PROGRAM POU
VAR
    fbDALI102Off             : FB_DALI102Off(POU_Comm.fbKL6821Communication);
    fbDALI102Off1            : FB_DALI102Off(POU_Comm.fbKL6821Communication);
    fbDALI102Off2            : FB_DALI102Off(POU_Comm.fbKL6821Communication);
    fbDALI102Off3            : FB_DALI102Off(POU_Comm.fbKL6821Communication);
    fbDALI102Dimmer1Switch   : FB_DALI102Dimmer1Switch(POU_Comm.fbKL6821Communication);
    fbDALI102Dimmer2Switch   : FB_DALI102Dimmer1Switch(POU_Comm.fbKL6821Communication);
    fbDALI102Dimmer3Switch   : FB_DALI102Dimmer1Switch(POU_Comm.fbKL6821Communication);
    fbDALI102Dimmer4Switch   : FB_DALI102Dimmer1Switch(POU_Comm.fbKL6821Communication);
    fbDALI102Dimmer5Switch   : FB_DALI102Dimmer1Switch(POU_Comm.fbKL6821Communication);
    fbDALI102Dimmer6Switch   : FB_DALI102Dimmer1Switch(POU_Comm.fbKL6821Communication);
    fbDALI102Dimmer7Switch   : FB_DALI102Dimmer1Switch(POU_Comm.fbKL6821Communication);
    fbDALI102Dimmer8Switch   : FB_DALI102Dimmer1Switch(POU_Comm.fbKL6821Communication);
    fbDALI102Dimmer9Switch   : FB_DALI102Dimmer1Switch(POU_Comm.fbKL6821Communication);
    fbDALI102Dimmer10Switch  : FB_DALI102Dimmer1Switch(POU_Comm.fbKL6821Communication);
    fbDALI102Dimmer11Switch  : FB_DALI102Dimmer1Switch(POU_Comm.fbKL6821Communication);
    fbDALI102Dimmer12Switch  : FB_DALI102Dimmer1Switch(POU_Comm.fbKL6821Communication);
    fbDALI102Dimmer13Switch  : FB_DALI102Dimmer1Switch(POU_Comm.fbKL6821Communication);
    fbDALI102Dimmer14Switch  : FB_DALI102Dimmer1Switch(POU_Comm.fbKL6821Communication);
    fbDALI102Dimmer15Switch  : FB_DALI102Dimmer1Switch(POU_Comm.fbKL6821Communication);
    fbDALI102Dimmer16Switch  : FB_DALI102Dimmer1Switch(POU_Comm.fbKL6821Communication);
    fbDALI102Dimmer17Switch  : FB_DALI102Dimmer1Switch(POU_Comm.fbKL6821Communication);
    fbDALI102Dimmer18Switch  : FB_DALI102Dimmer1Switch(POU_Comm.fbKL6821Communication);
    fbDALI102Dimmer19Switch  : FB_DALI102Dimmer1Switch(POU_Comm.fbKL6821Communication);
    fbDALI102Dimmer20Switch  : FB_DALI102Dimmer1Switch(POU_Comm.fbKL6821Communication);
    fbDALI102Dimmer21Switch  : FB_DALI102Dimmer1Switch(POU_Comm.fbKL6821Communication);
    fbDALI102Dimmer22Switch  : FB_DALI102Dimmer1Switch(POU_Comm.fbKL6821Communication);
    fbDALI102Dimmer23Switch  : FB_DALI102Dimmer1Switch(POU_Comm.fbKL6821Communication);
    fbDALI102Dimmer24Switch  : FB_DALI102Dimmer1Switch(POU_Comm.fbKL6821Communication);
    fbDALI102Dimmer25Switch  : FB_DALI102Dimmer1Switch(POU_Comm.fbKL6821Communication);
    fbDALI102Dimmer26Switch  : FB_DALI102Dimmer1Switch(POU_Comm.fbKL6821Communication);
    fbDALI102Dimmer27Switch  : FB_DALI102Dimmer1Switch(POU_Comm.fbKL6821Communication);
    fbDALI102Dimmer28Switch  : FB_DALI102Dimmer1Switch(POU_Comm.fbKL6821Communication);
    bInitialize              : BOOL := FALSE;
    motionSensor             : BOOL;
    bRecallMaxLevel          : BOOL;
    bRecallMinLevel          : BOOL;
    bToggle                  : BOOL;
    bGoToScene               : BOOL;
    nScene                   : BYTE;
    bSetLevel                : BOOL;
    nLevel                   : BYTE := 254;
    nLevelMemoryMode         : BYTE := 254;
    nReferenceDeviceAddress  : BYTE;
    tCycleActualLevel        : TIME := T#5S;
    nOptions                 : DWORD := 0;
    nActualLevel             : BYTE;
END_VAR

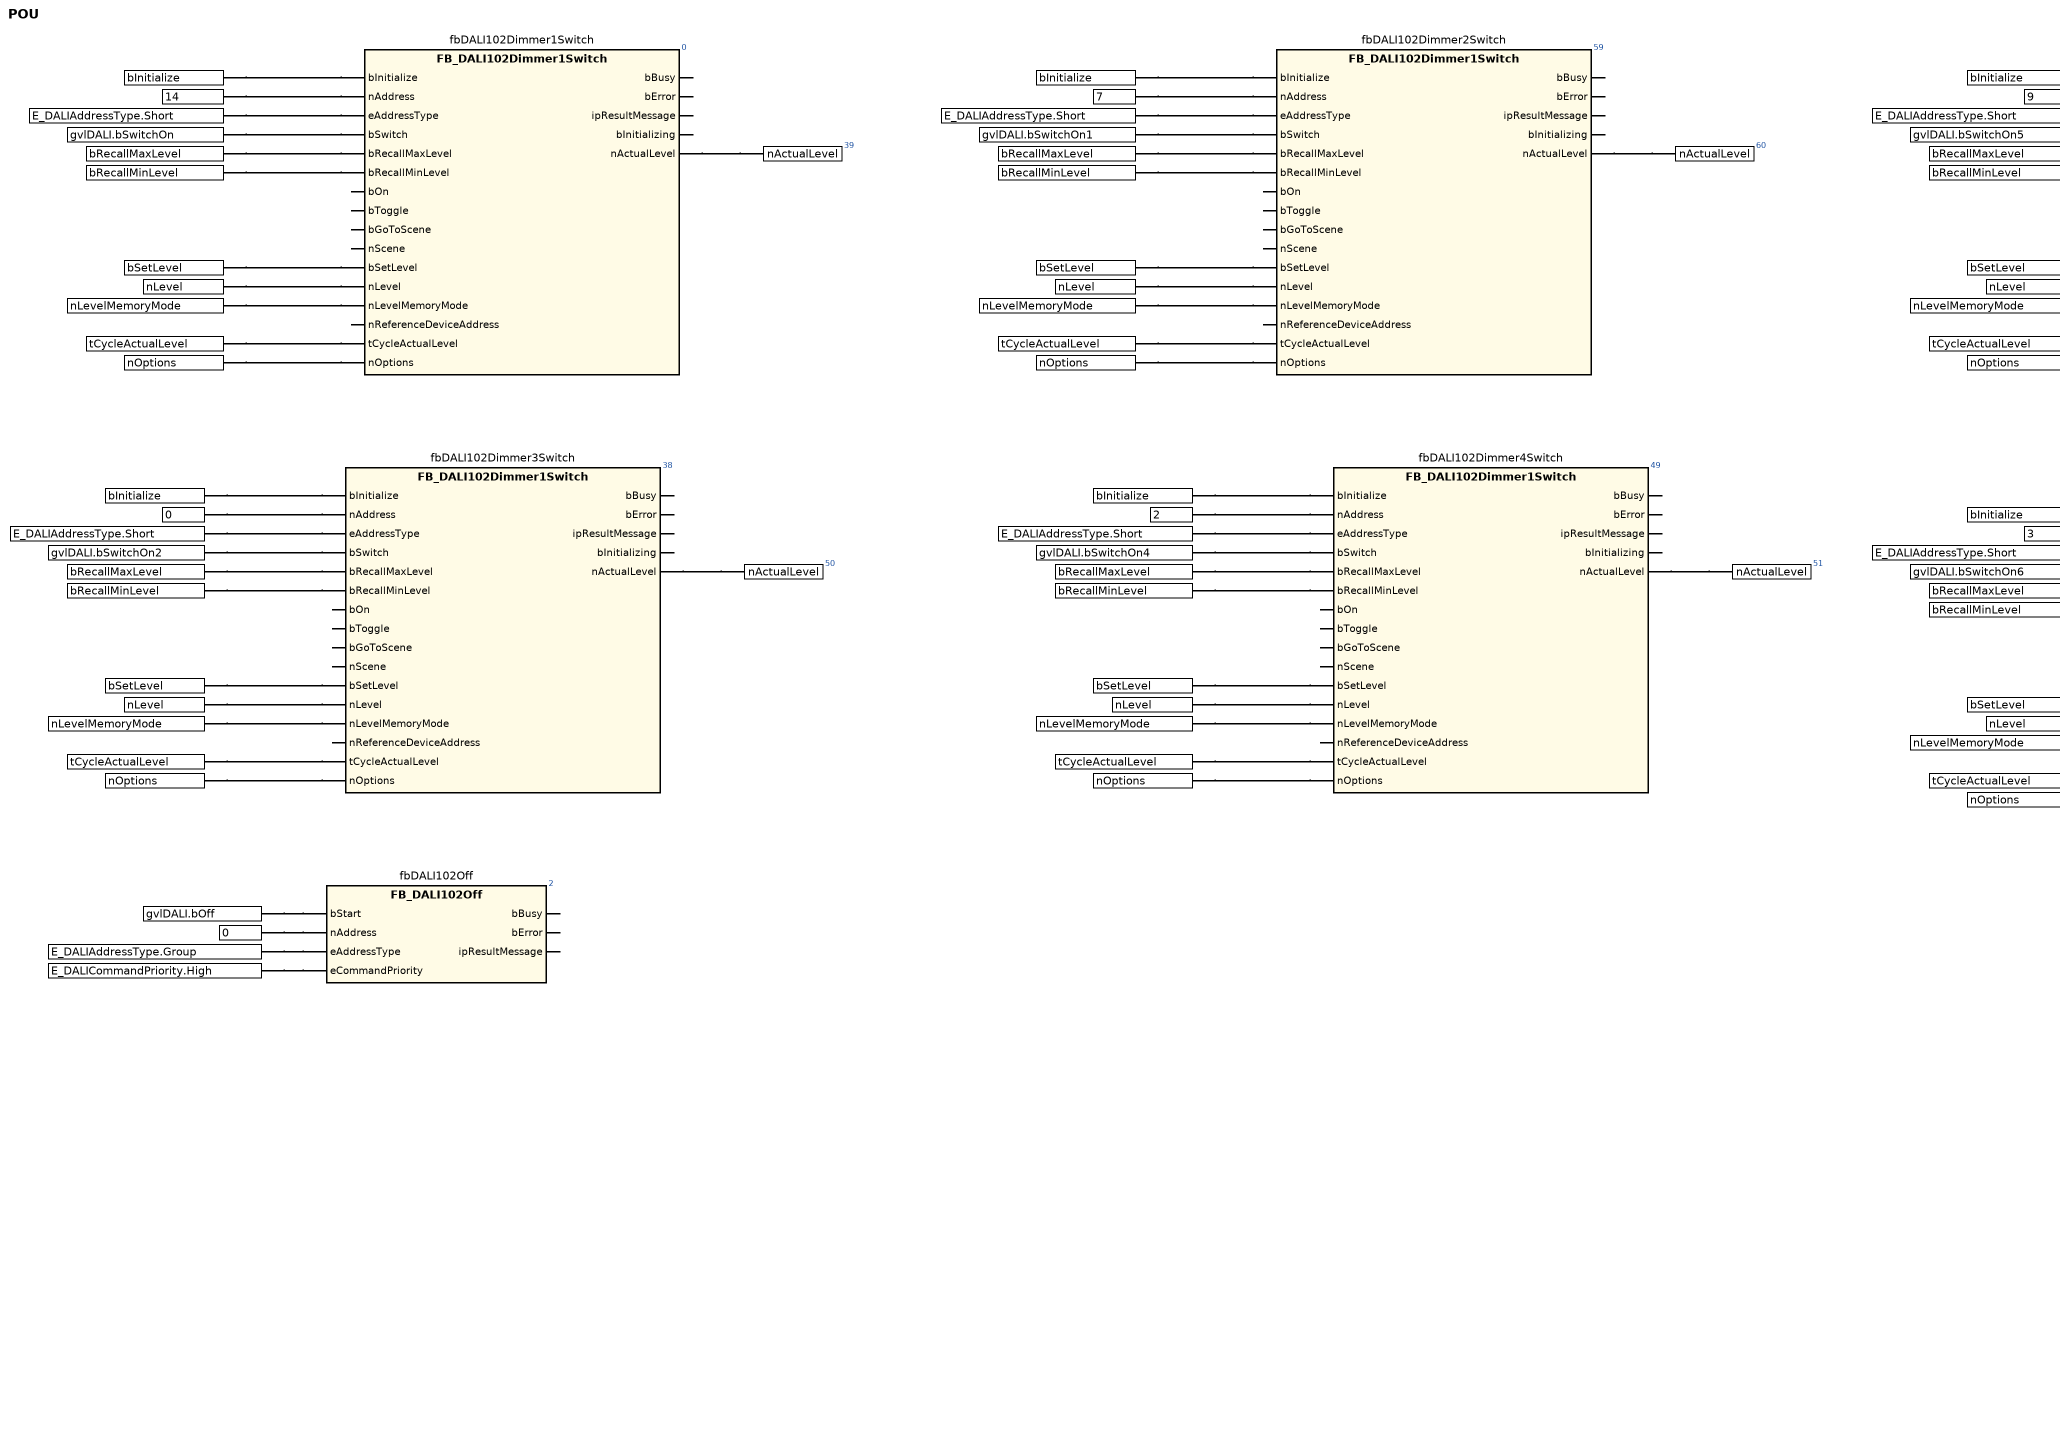
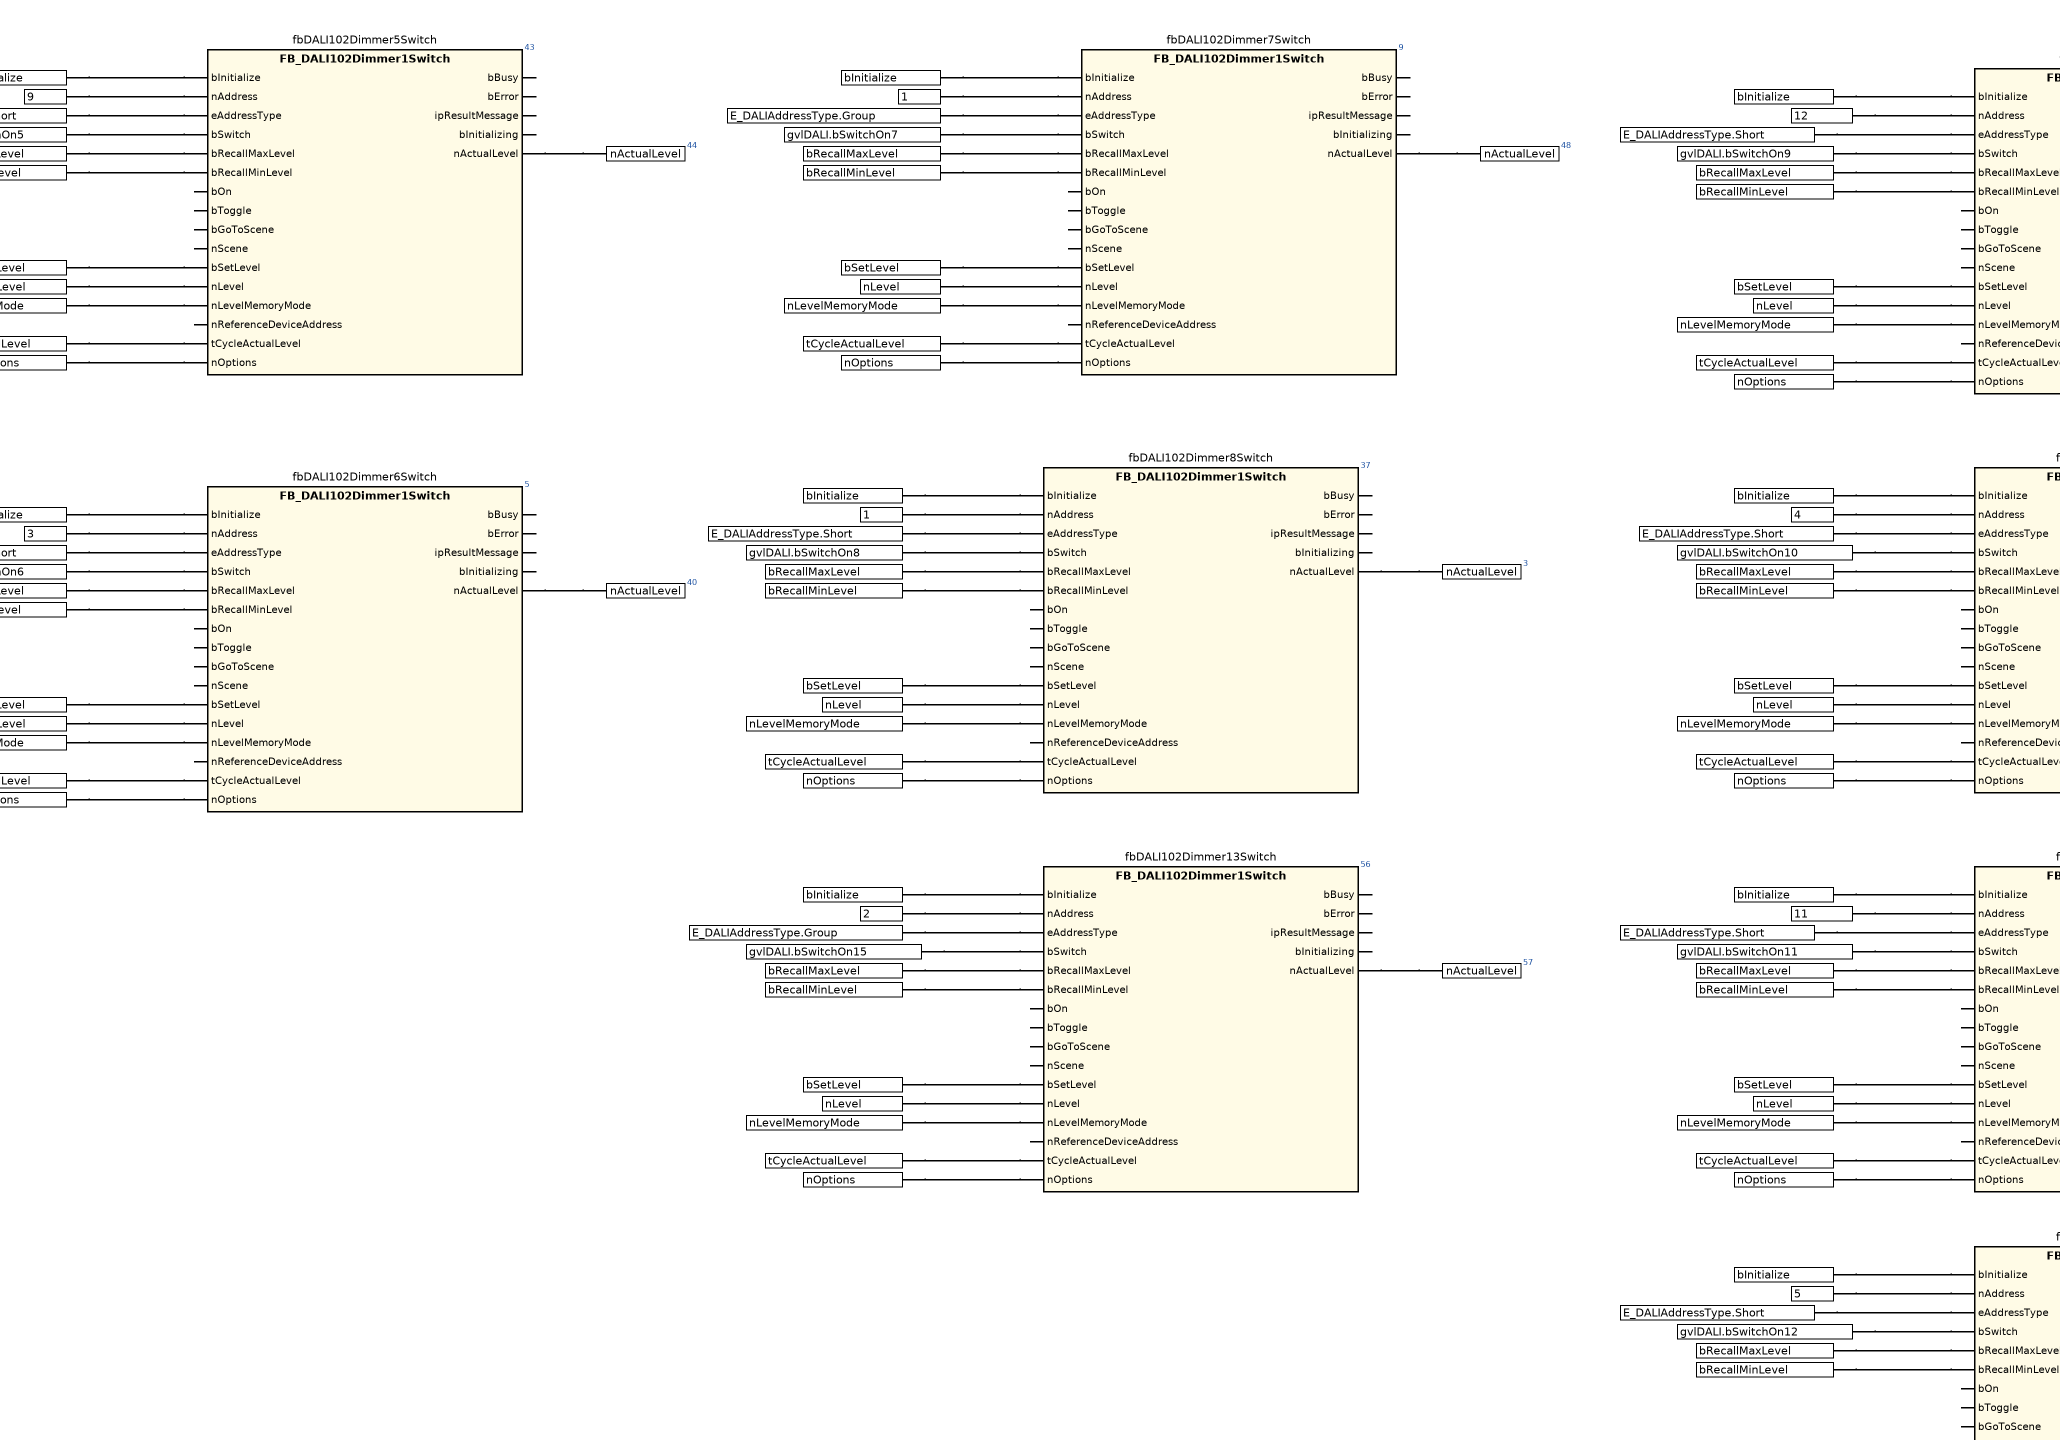
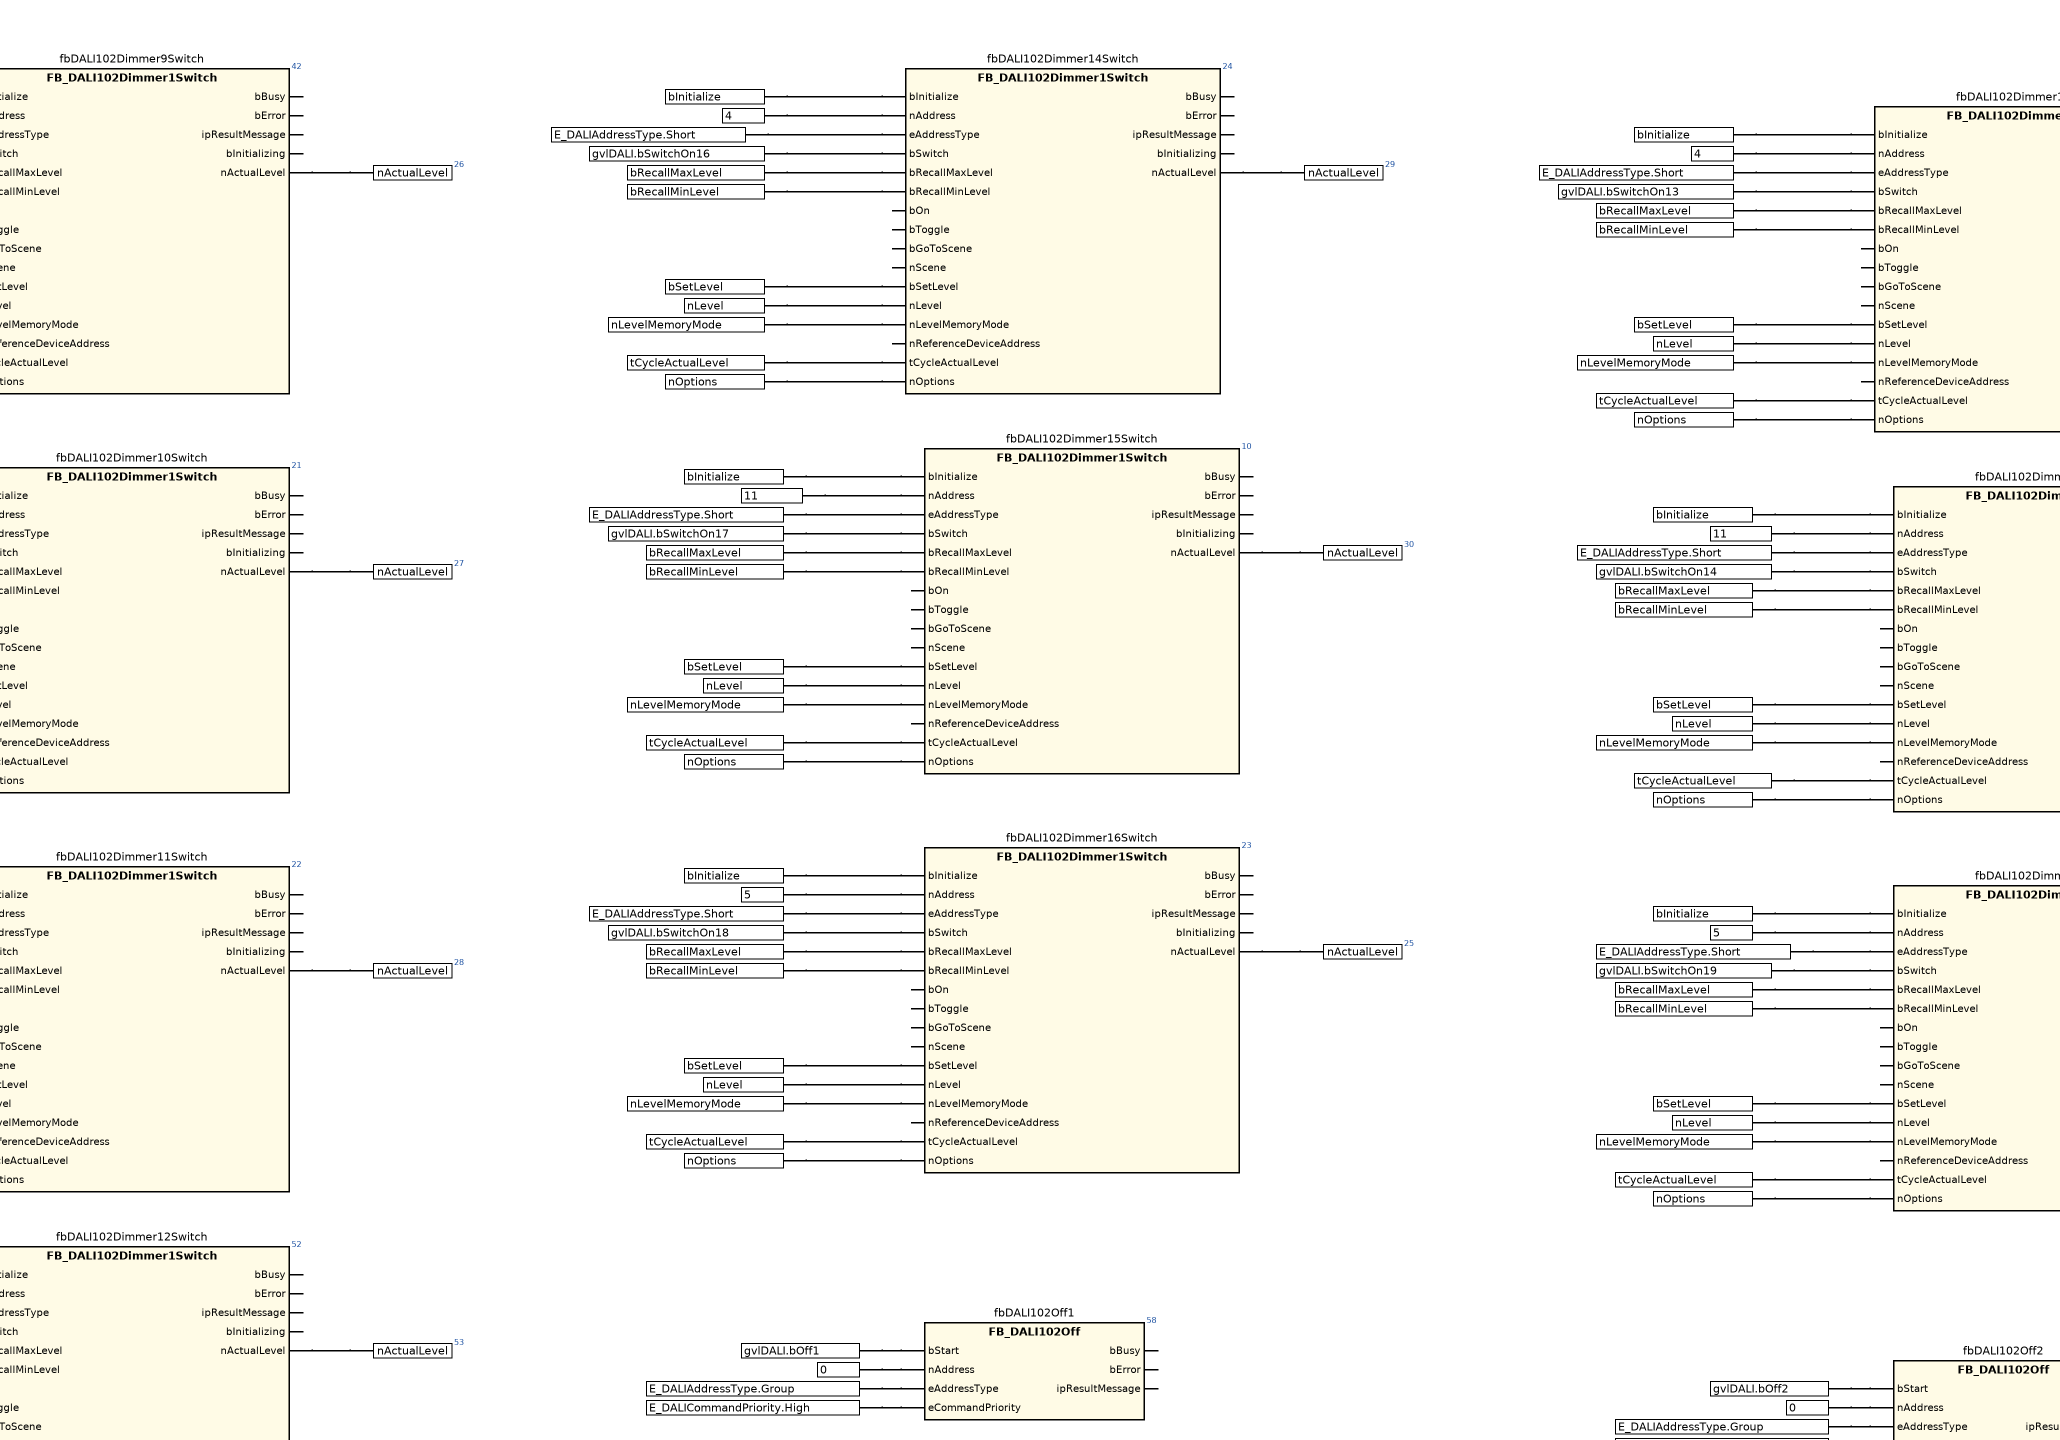
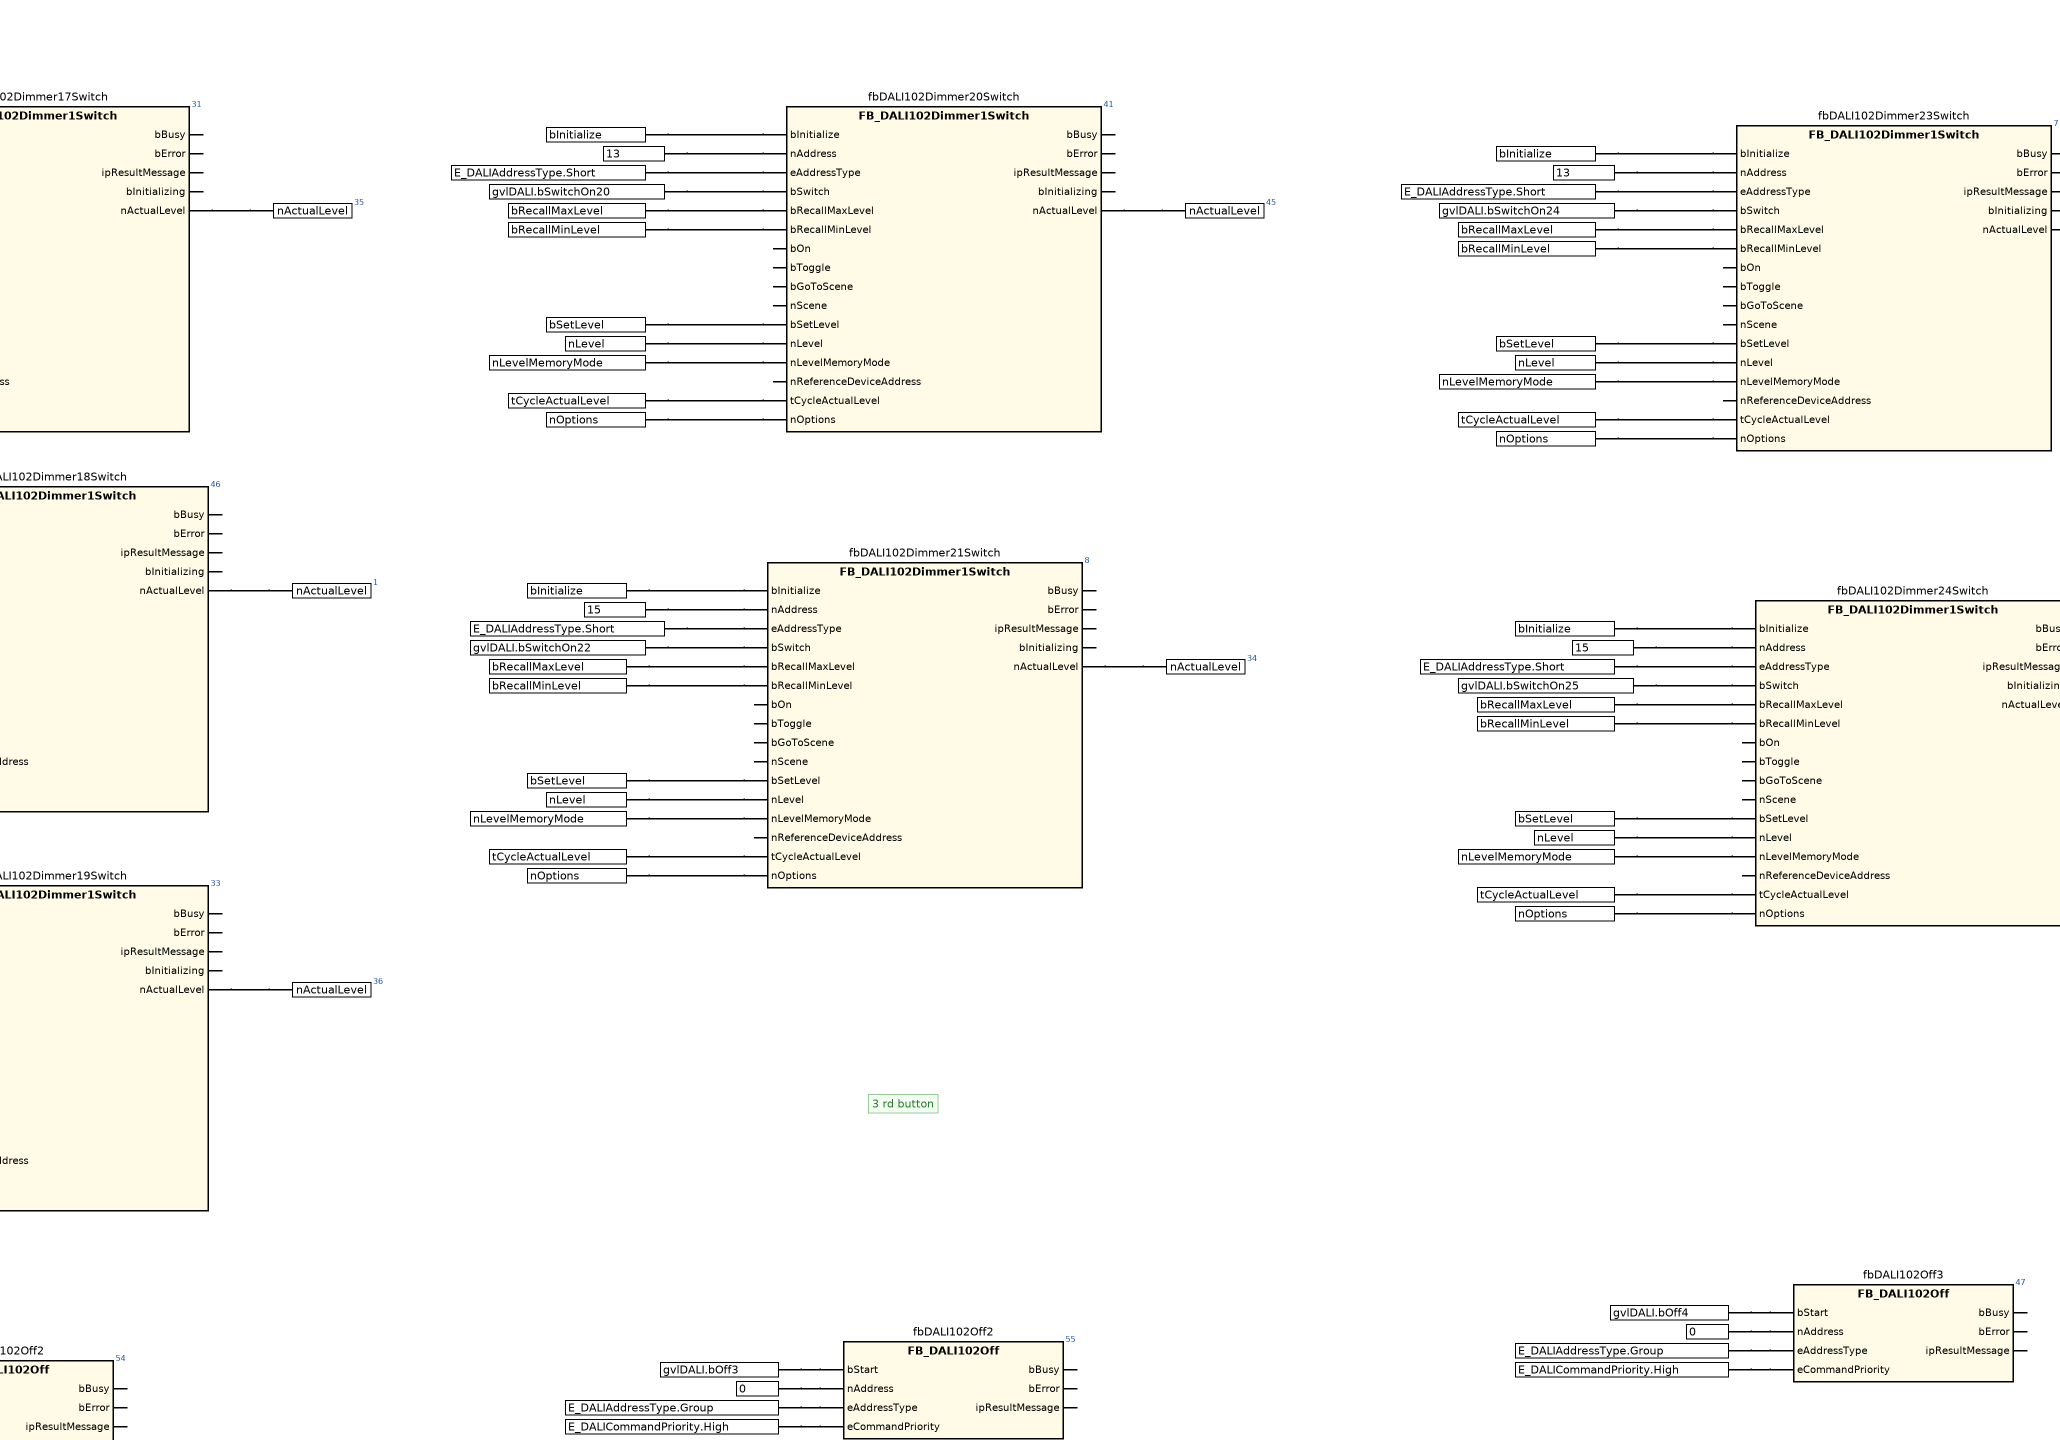
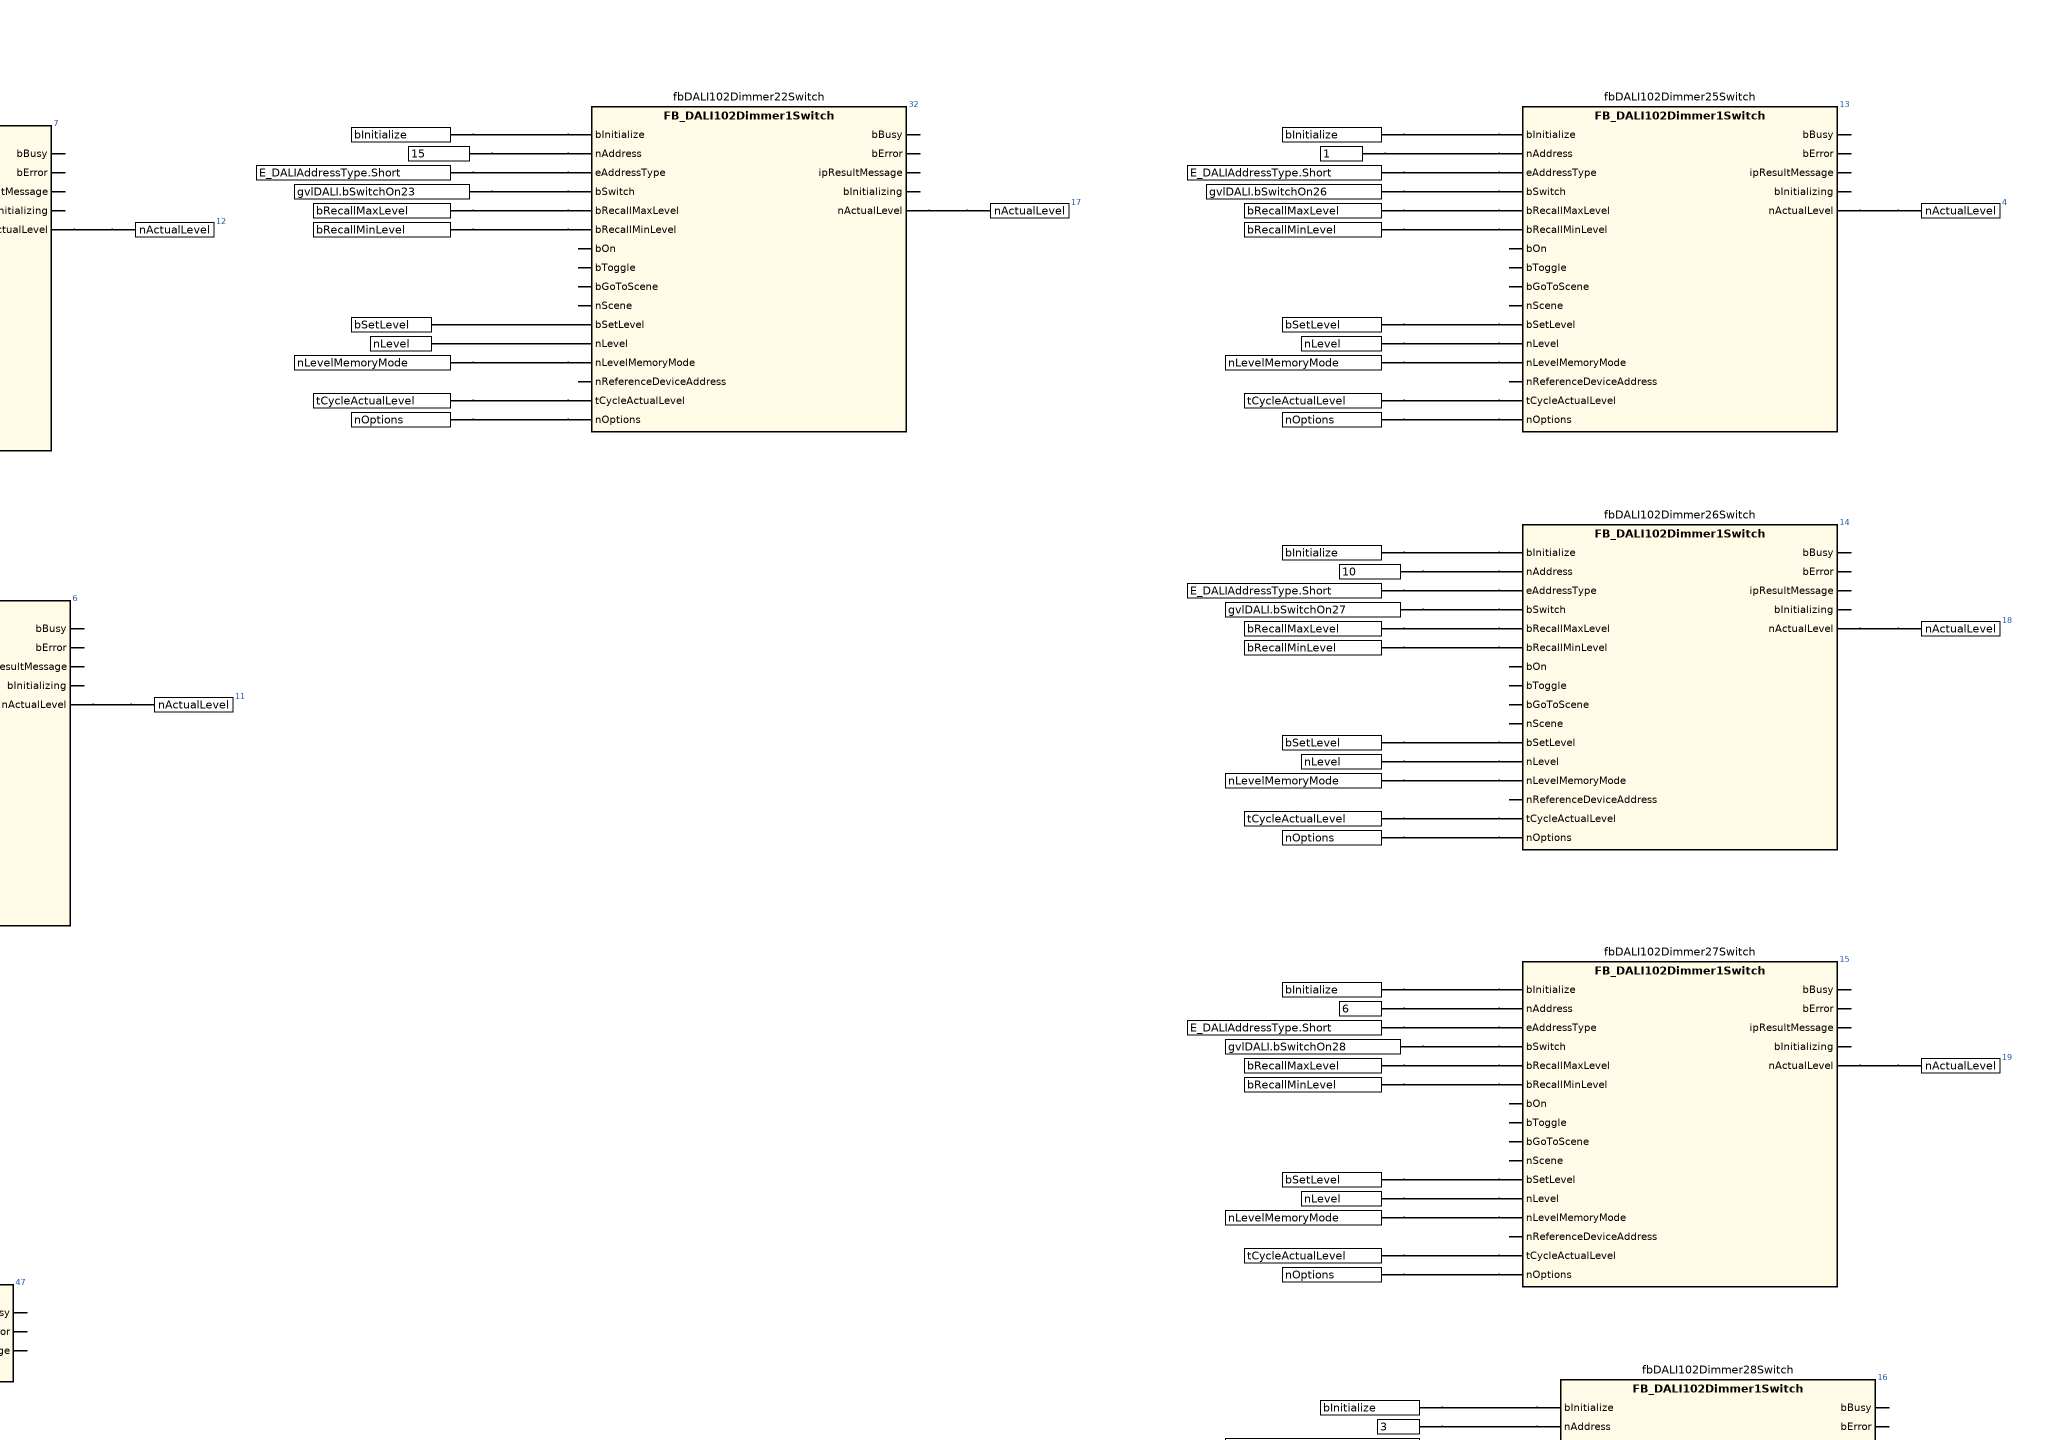
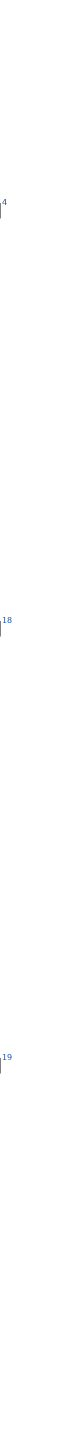
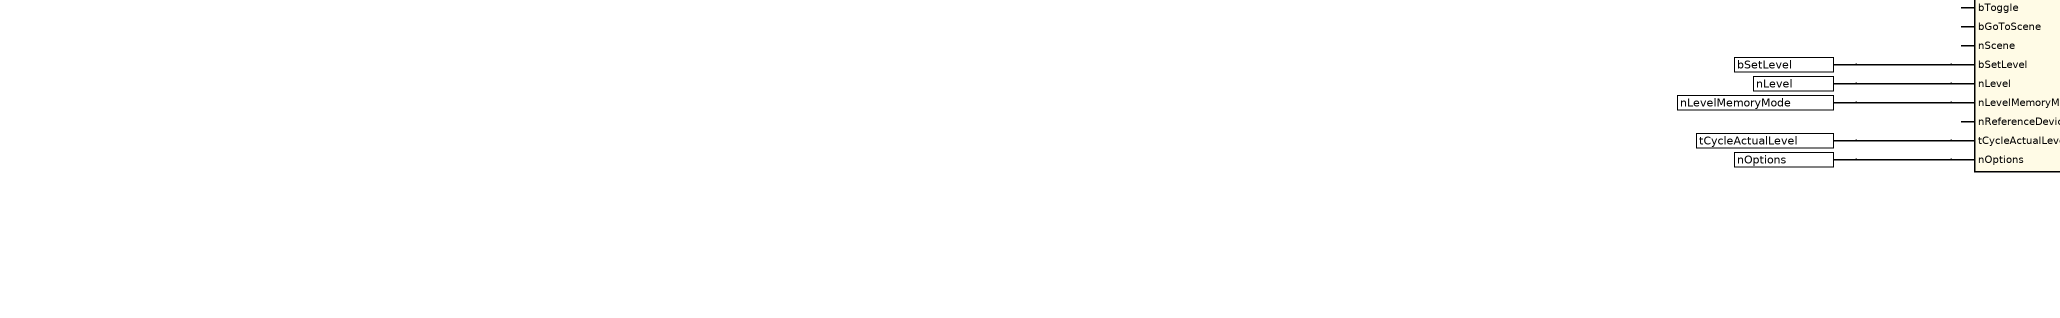
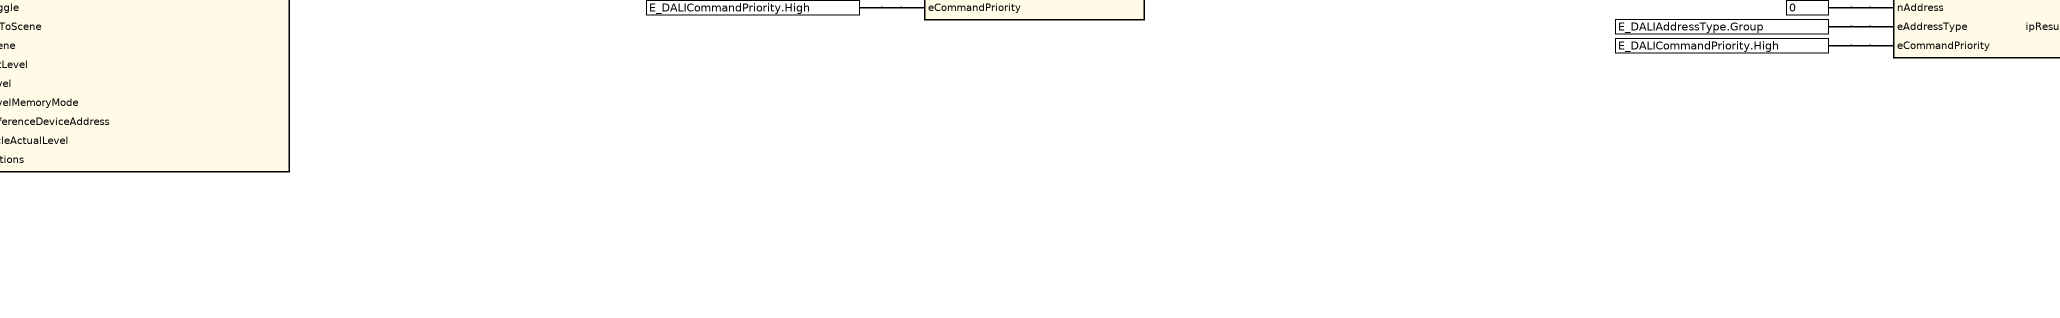
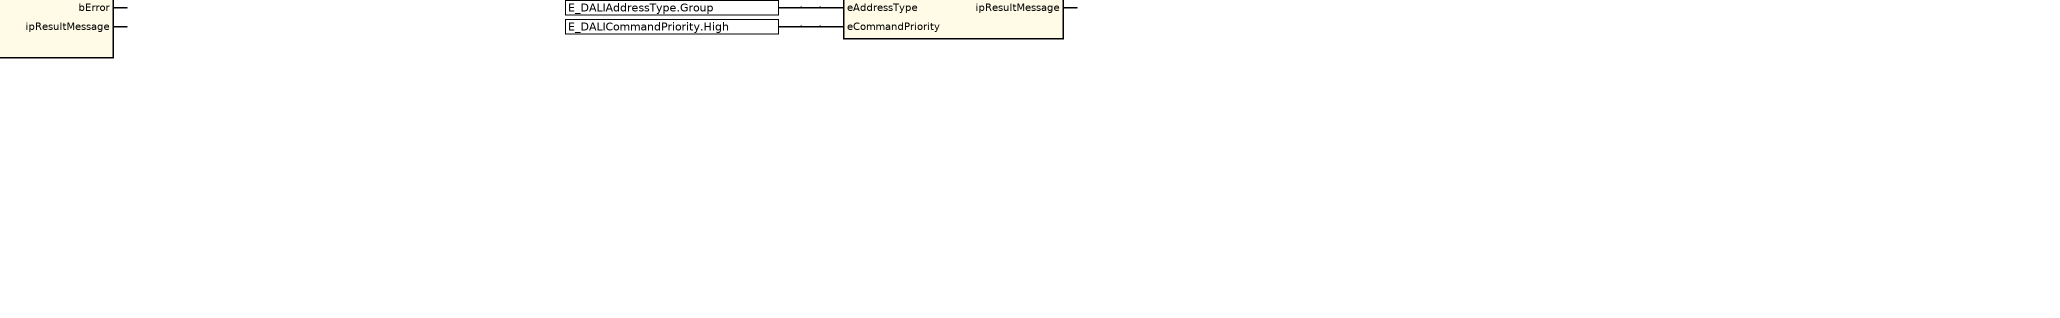
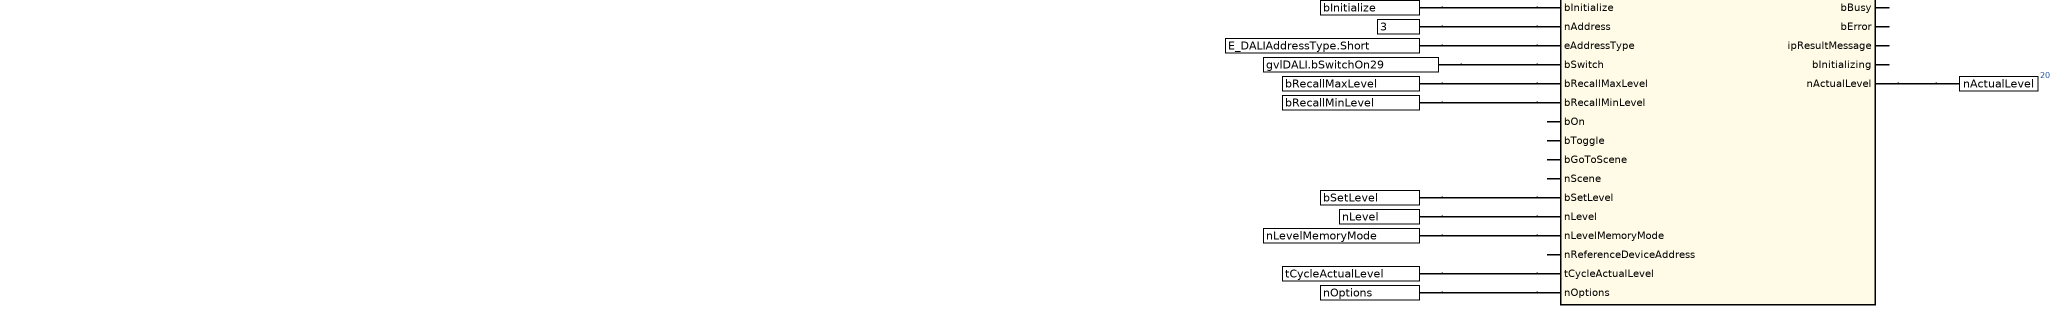
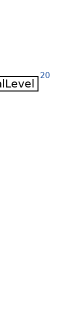
fbDALI102Dimmer1Switch(
    bInitialize := bInitialize,
    nAddress := 14,
    eAddressType := E_DALIAddressType.Short,
    bSwitch := gvlDALI.bSwitchOn,
    bRecallMaxLevel := bRecallMaxLevel,
    bRecallMinLevel := bRecallMinLevel,
    bSetLevel := bSetLevel,
    nLevel := nLevel,
    nLevelMemoryMode := nLevelMemoryMode,
    tCycleActualLevel := tCycleActualLevel,
    nOptions := nOptions); // FB_DALI102Dimmer1Switch
nActualLevel := fbDALI102Dimmer18Switch.nActualLevel;
fbDALI102Off(
    bStart := gvlDALI.bOff,
    nAddress := 0,
    eAddressType := E_DALIAddressType.Group,
    eCommandPriority := E_DALICommandPriority.High); // FB_DALI102Off
nActualLevel := fbDALI102Dimmer8Switch.nActualLevel;
nActualLevel := fbDALI102Dimmer25Switch.nActualLevel;
fbDALI102Dimmer6Switch(
    bInitialize := bInitialize,
    nAddress := 3,
    eAddressType := E_DALIAddressType.Short,
    bSwitch := gvlDALI.bSwitchOn6,
    bRecallMaxLevel := bRecallMaxLevel,
    bRecallMinLevel := bRecallMinLevel,
    bSetLevel := bSetLevel,
    nLevel := nLevel,
    nLevelMemoryMode := nLevelMemoryMode,
    tCycleActualLevel := tCycleActualLevel,
    nOptions := nOptions); // FB_DALI102Dimmer1Switch
fbDALI102Dimmer24Switch(
    bInitialize := bInitialize,
    nAddress := 15,
    eAddressType := E_DALIAddressType.Short,
    bSwitch := gvlDALI.bSwitchOn25,
    bRecallMaxLevel := bRecallMaxLevel,
    bRecallMinLevel := bRecallMinLevel,
    bSetLevel := bSetLevel,
    nLevel := nLevel,
    nLevelMemoryMode := nLevelMemoryMode,
    tCycleActualLevel := tCycleActualLevel,
    nOptions := nOptions); // FB_DALI102Dimmer1Switch
fbDALI102Dimmer23Switch(
    bInitialize := bInitialize,
    nAddress := 13,
    eAddressType := E_DALIAddressType.Short,
    bSwitch := gvlDALI.bSwitchOn24,
    bRecallMaxLevel := bRecallMaxLevel,
    bRecallMinLevel := bRecallMinLevel,
    bSetLevel := bSetLevel,
    nLevel := nLevel,
    nLevelMemoryMode := nLevelMemoryMode,
    tCycleActualLevel := tCycleActualLevel,
    nOptions := nOptions); // FB_DALI102Dimmer1Switch
fbDALI102Dimmer21Switch(
    bInitialize := bInitialize,
    nAddress := 15,
    eAddressType := E_DALIAddressType.Short,
    bSwitch := gvlDALI.bSwitchOn22,
    bRecallMaxLevel := bRecallMaxLevel,
    bRecallMinLevel := bRecallMinLevel,
    bSetLevel := bSetLevel,
    nLevel := nLevel,
    nLevelMemoryMode := nLevelMemoryMode,
    tCycleActualLevel := tCycleActualLevel,
    nOptions := nOptions); // FB_DALI102Dimmer1Switch
fbDALI102Dimmer7Switch(
    bInitialize := bInitialize,
    nAddress := 1,
    eAddressType := E_DALIAddressType.Group,
    bSwitch := gvlDALI.bSwitchOn7,
    bRecallMaxLevel := bRecallMaxLevel,
    bRecallMinLevel := bRecallMinLevel,
    bSetLevel := bSetLevel,
    nLevel := nLevel,
    nLevelMemoryMode := nLevelMemoryMode,
    tCycleActualLevel := tCycleActualLevel,
    nOptions := nOptions); // FB_DALI102Dimmer1Switch
fbDALI102Dimmer15Switch(
    bInitialize := bInitialize,
    nAddress := 11,
    eAddressType := E_DALIAddressType.Short,
    bSwitch := gvlDALI.bSwitchOn17,
    bRecallMaxLevel := bRecallMaxLevel,
    bRecallMinLevel := bRecallMinLevel,
    bSetLevel := bSetLevel,
    nLevel := nLevel,
    nLevelMemoryMode := nLevelMemoryMode,
    tCycleActualLevel := tCycleActualLevel,
    nOptions := nOptions); // FB_DALI102Dimmer1Switch
nActualLevel := fbDALI102Dimmer24Switch.nActualLevel;
nActualLevel := fbDALI102Dimmer23Switch.nActualLevel;
fbDALI102Dimmer25Switch(
    bInitialize := bInitialize,
    nAddress := 1,
    eAddressType := E_DALIAddressType.Short,
    bSwitch := gvlDALI.bSwitchOn26,
    bRecallMaxLevel := bRecallMaxLevel,
    bRecallMinLevel := bRecallMinLevel,
    bSetLevel := bSetLevel,
    nLevel := nLevel,
    nLevelMemoryMode := nLevelMemoryMode,
    tCycleActualLevel := tCycleActualLevel,
    nOptions := nOptions); // FB_DALI102Dimmer1Switch
fbDALI102Dimmer26Switch(
    bInitialize := bInitialize,
    nAddress := 10,
    eAddressType := E_DALIAddressType.Short,
    bSwitch := gvlDALI.bSwitchOn27,
    bRecallMaxLevel := bRecallMaxLevel,
    bRecallMinLevel := bRecallMinLevel,
    bSetLevel := bSetLevel,
    nLevel := nLevel,
    nLevelMemoryMode := nLevelMemoryMode,
    tCycleActualLevel := tCycleActualLevel,
    nOptions := nOptions); // FB_DALI102Dimmer1Switch
fbDALI102Dimmer27Switch(
    bInitialize := bInitialize,
    nAddress := 6,
    eAddressType := E_DALIAddressType.Short,
    bSwitch := gvlDALI.bSwitchOn28,
    bRecallMaxLevel := bRecallMaxLevel,
    bRecallMinLevel := bRecallMinLevel,
    bSetLevel := bSetLevel,
    nLevel := nLevel,
    nLevelMemoryMode := nLevelMemoryMode,
    tCycleActualLevel := tCycleActualLevel,
    nOptions := nOptions); // FB_DALI102Dimmer1Switch
fbDALI102Dimmer28Switch(
    bInitialize := bInitialize,
    nAddress := 3,
    eAddressType := E_DALIAddressType.Short,
    bSwitch := gvlDALI.bSwitchOn29,
    bRecallMaxLevel := bRecallMaxLevel,
    bRecallMinLevel := bRecallMinLevel,
    bSetLevel := bSetLevel,
    nLevel := nLevel,
    nLevelMemoryMode := nLevelMemoryMode,
    tCycleActualLevel := tCycleActualLevel,
    nOptions := nOptions); // FB_DALI102Dimmer1Switch
nActualLevel := fbDALI102Dimmer22Switch.nActualLevel;
nActualLevel := fbDALI102Dimmer26Switch.nActualLevel;
nActualLevel := fbDALI102Dimmer27Switch.nActualLevel;
nActualLevel := fbDALI102Dimmer28Switch.nActualLevel;
fbDALI102Dimmer10Switch(
    bInitialize := bInitialize,
    nAddress := 4,
    eAddressType := E_DALIAddressType.Short,
    bSwitch := gvlDALI.bSwitchOn10,
    bRecallMaxLevel := bRecallMaxLevel,
    bRecallMinLevel := bRecallMinLevel,
    bSetLevel := bSetLevel,
    nLevel := nLevel,
    nLevelMemoryMode := nLevelMemoryMode,
    tCycleActualLevel := tCycleActualLevel,
    nOptions := nOptions); // FB_DALI102Dimmer1Switch
fbDALI102Dimmer11Switch(
    bInitialize := bInitialize,
    nAddress := 11,
    eAddressType := E_DALIAddressType.Short,
    bSwitch := gvlDALI.bSwitchOn11,
    bRecallMaxLevel := bRecallMaxLevel,
    bRecallMinLevel := bRecallMinLevel,
    bSetLevel := bSetLevel,
    nLevel := nLevel,
    nLevelMemoryMode := nLevelMemoryMode,
    tCycleActualLevel := tCycleActualLevel,
    nOptions := nOptions); // FB_DALI102Dimmer1Switch
fbDALI102Dimmer16Switch(
    bInitialize := bInitialize,
    nAddress := 5,
    eAddressType := E_DALIAddressType.Short,
    bSwitch := gvlDALI.bSwitchOn18,
    bRecallMaxLevel := bRecallMaxLevel,
    bRecallMinLevel := bRecallMinLevel,
    bSetLevel := bSetLevel,
    nLevel := nLevel,
    nLevelMemoryMode := nLevelMemoryMode,
    tCycleActualLevel := tCycleActualLevel,
    nOptions := nOptions); // FB_DALI102Dimmer1Switch
fbDALI102Dimmer14Switch(
    bInitialize := bInitialize,
    nAddress := 4,
    eAddressType := E_DALIAddressType.Short,
    bSwitch := gvlDALI.bSwitchOn16,
    bRecallMaxLevel := bRecallMaxLevel,
    bRecallMinLevel := bRecallMinLevel,
    bSetLevel := bSetLevel,
    nLevel := nLevel,
    nLevelMemoryMode := nLevelMemoryMode,
    tCycleActualLevel := tCycleActualLevel,
    nOptions := nOptions); // FB_DALI102Dimmer1Switch
nActualLevel := fbDALI102Dimmer16Switch.nActualLevel;
nActualLevel := fbDALI102Dimmer9Switch.nActualLevel;
nActualLevel := fbDALI102Dimmer10Switch.nActualLevel;
nActualLevel := fbDALI102Dimmer11Switch.nActualLevel;
nActualLevel := fbDALI102Dimmer14Switch.nActualLevel;
nActualLevel := fbDALI102Dimmer15Switch.nActualLevel;
fbDALI102Dimmer17Switch(
    bInitialize := bInitialize,
    nAddress := 4,
    eAddressType := E_DALIAddressType.Short,
    bSwitch := gvlDALI.bSwitchOn13,
    bRecallMaxLevel := bRecallMaxLevel,
    bRecallMinLevel := bRecallMinLevel,
    bSetLevel := bSetLevel,
    nLevel := nLevel,
    nLevelMemoryMode := nLevelMemoryMode,
    tCycleActualLevel := tCycleActualLevel,
    nOptions := nOptions); // FB_DALI102Dimmer1Switch
fbDALI102Dimmer22Switch(
    bInitialize := bInitialize,
    nAddress := 15,
    eAddressType := E_DALIAddressType.Short,
    bSwitch := gvlDALI.bSwitchOn23,
    bRecallMaxLevel := bRecallMaxLevel,
    bRecallMinLevel := bRecallMinLevel,
    bSetLevel := bSetLevel,
    nLevel := nLevel,
    nLevelMemoryMode := nLevelMemoryMode,
    tCycleActualLevel := tCycleActualLevel,
    nOptions := nOptions); // FB_DALI102Dimmer1Switch
fbDALI102Dimmer19Switch(
    bInitialize := bInitialize,
    nAddress := 5,
    eAddressType := E_DALIAddressType.Short,
    bSwitch := gvlDALI.bSwitchOn19,
    bRecallMaxLevel := bRecallMaxLevel,
    bRecallMinLevel := bRecallMinLevel,
    bSetLevel := bSetLevel,
    nLevel := nLevel,
    nLevelMemoryMode := nLevelMemoryMode,
    tCycleActualLevel := tCycleActualLevel,
    nOptions := nOptions); // FB_DALI102Dimmer1Switch
nActualLevel := fbDALI102Dimmer21Switch.nActualLevel;
nActualLevel := fbDALI102Dimmer17Switch.nActualLevel;
nActualLevel := fbDALI102Dimmer19Switch.nActualLevel;
fbDALI102Dimmer8Switch(
    bInitialize := bInitialize,
    nAddress := 1,
    eAddressType := E_DALIAddressType.Short,
    bSwitch := gvlDALI.bSwitchOn8,
    bRecallMaxLevel := bRecallMaxLevel,
    bRecallMinLevel := bRecallMinLevel,
    bSetLevel := bSetLevel,
    nLevel := nLevel,
    nLevelMemoryMode := nLevelMemoryMode,
    tCycleActualLevel := tCycleActualLevel,
    nOptions := nOptions); // FB_DALI102Dimmer1Switch
fbDALI102Dimmer3Switch(
    bInitialize := bInitialize,
    nAddress := 0,
    eAddressType := E_DALIAddressType.Short,
    bSwitch := gvlDALI.bSwitchOn2,
    bRecallMaxLevel := bRecallMaxLevel,
    bRecallMinLevel := bRecallMinLevel,
    bSetLevel := bSetLevel,
    nLevel := nLevel,
    nLevelMemoryMode := nLevelMemoryMode,
    tCycleActualLevel := tCycleActualLevel,
    nOptions := nOptions); // FB_DALI102Dimmer1Switch
nActualLevel := fbDALI102Dimmer1Switch.nActualLevel;
nActualLevel := fbDALI102Dimmer6Switch.nActualLevel;
fbDALI102Dimmer20Switch(
    bInitialize := bInitialize,
    nAddress := 13,
    eAddressType := E_DALIAddressType.Short,
    bSwitch := gvlDALI.bSwitchOn20,
    bRecallMaxLevel := bRecallMaxLevel,
    bRecallMinLevel := bRecallMinLevel,
    bSetLevel := bSetLevel,
    nLevel := nLevel,
    nLevelMemoryMode := nLevelMemoryMode,
    tCycleActualLevel := tCycleActualLevel,
    nOptions := nOptions); // FB_DALI102Dimmer1Switch
fbDALI102Dimmer9Switch(
    bInitialize := bInitialize,
    nAddress := 12,
    eAddressType := E_DALIAddressType.Short,
    bSwitch := gvlDALI.bSwitchOn9,
    bRecallMaxLevel := bRecallMaxLevel,
    bRecallMinLevel := bRecallMinLevel,
    bSetLevel := bSetLevel,
    nLevel := nLevel,
    nLevelMemoryMode := nLevelMemoryMode,
    tCycleActualLevel := tCycleActualLevel,
    nOptions := nOptions); // FB_DALI102Dimmer1Switch
fbDALI102Dimmer5Switch(
    bInitialize := bInitialize,
    nAddress := 9,
    eAddressType := E_DALIAddressType.Short,
    bSwitch := gvlDALI.bSwitchOn5,
    bRecallMaxLevel := bRecallMaxLevel,
    bRecallMinLevel := bRecallMinLevel,
    bSetLevel := bSetLevel,
    nLevel := nLevel,
    nLevelMemoryMode := nLevelMemoryMode,
    tCycleActualLevel := tCycleActualLevel,
    nOptions := nOptions); // FB_DALI102Dimmer1Switch
nActualLevel := fbDALI102Dimmer5Switch.nActualLevel;
nActualLevel := fbDALI102Dimmer20Switch.nActualLevel;
fbDALI102Dimmer18Switch(
    bInitialize := bInitialize,
    nAddress := 11,
    eAddressType := E_DALIAddressType.Short,
    bSwitch := gvlDALI.bSwitchOn14,
    bRecallMaxLevel := bRecallMaxLevel,
    bRecallMinLevel := bRecallMinLevel,
    bSetLevel := bSetLevel,
    nLevel := nLevel,
    nLevelMemoryMode := nLevelMemoryMode,
    tCycleActualLevel := tCycleActualLevel,
    nOptions := nOptions); // FB_DALI102Dimmer1Switch
fbDALI102Off3(
    bStart := gvlDALI.bOff4,
    nAddress := 0,
    eAddressType := E_DALIAddressType.Group,
    eCommandPriority := E_DALICommandPriority.High); // FB_DALI102Off
nActualLevel := fbDALI102Dimmer7Switch.nActualLevel;
fbDALI102Dimmer4Switch(
    bInitialize := bInitialize,
    nAddress := 2,
    eAddressType := E_DALIAddressType.Short,
    bSwitch := gvlDALI.bSwitchOn4,
    bRecallMaxLevel := bRecallMaxLevel,
    bRecallMinLevel := bRecallMinLevel,
    bSetLevel := bSetLevel,
    nLevel := nLevel,
    nLevelMemoryMode := nLevelMemoryMode,
    tCycleActualLevel := tCycleActualLevel,
    nOptions := nOptions); // FB_DALI102Dimmer1Switch
nActualLevel := fbDALI102Dimmer3Switch.nActualLevel;
nActualLevel := fbDALI102Dimmer4Switch.nActualLevel;
fbDALI102Dimmer12Switch(
    bInitialize := bInitialize,
    nAddress := 5,
    eAddressType := E_DALIAddressType.Short,
    bSwitch := gvlDALI.bSwitchOn12,
    bRecallMaxLevel := bRecallMaxLevel,
    bRecallMinLevel := bRecallMinLevel,
    bSetLevel := bSetLevel,
    nLevel := nLevel,
    nLevelMemoryMode := nLevelMemoryMode,
    tCycleActualLevel := tCycleActualLevel,
    nOptions := nOptions); // FB_DALI102Dimmer1Switch
nActualLevel := fbDALI102Dimmer12Switch.nActualLevel;
fbDALI102Off2(
    bStart := gvlDALI.bOff2,
    nAddress := 0,
    eAddressType := E_DALIAddressType.Group,
    eCommandPriority := E_DALICommandPriority.High); // FB_DALI102Off
// 3 rd button
fbDALI102Off2(
    bStart := gvlDALI.bOff3,
    nAddress := 0,
    eAddressType := E_DALIAddressType.Group,
    eCommandPriority := E_DALICommandPriority.High); // FB_DALI102Off
fbDALI102Dimmer13Switch(
    bInitialize := bInitialize,
    nAddress := 2,
    eAddressType := E_DALIAddressType.Group,
    bSwitch := gvlDALI.bSwitchOn15,
    bRecallMaxLevel := bRecallMaxLevel,
    bRecallMinLevel := bRecallMinLevel,
    bSetLevel := bSetLevel,
    nLevel := nLevel,
    nLevelMemoryMode := nLevelMemoryMode,
    tCycleActualLevel := tCycleActualLevel,
    nOptions := nOptions); // FB_DALI102Dimmer1Switch
nActualLevel := fbDALI102Dimmer13Switch.nActualLevel;
fbDALI102Off1(
    bStart := gvlDALI.bOff1,
    nAddress := 0,
    eAddressType := E_DALIAddressType.Group,
    eCommandPriority := E_DALICommandPriority.High); // FB_DALI102Off
fbDALI102Dimmer2Switch(
    bInitialize := bInitialize,
    nAddress := 7,
    eAddressType := E_DALIAddressType.Short,
    bSwitch := gvlDALI.bSwitchOn1,
    bRecallMaxLevel := bRecallMaxLevel,
    bRecallMinLevel := bRecallMinLevel,
    bSetLevel := bSetLevel,
    nLevel := nLevel,
    nLevelMemoryMode := nLevelMemoryMode,
    tCycleActualLevel := tCycleActualLevel,
    nOptions := nOptions); // FB_DALI102Dimmer1Switch
nActualLevel := fbDALI102Dimmer2Switch.nActualLevel;

END_PROGRAM

(* stored: Version 1.1.0.1, ProductVersion 3.1.4024.16
   POU POU: Id {f1177937-4de4-414d-9467-4ea23edb2c4f}, SpecialFunc None *)
